# EPICS substitutions: PicoscopeApp/Db/Picoscope.substitutions
file PicoscopeApp/Db/Picoscope.template
{
    pattern
    { channel }
    {    A    }
    {    B    }
    {    C    }
    {    D    }
}
